INTERFACE I_StepCondition

PROPERTY getValue : BOOL
GET
END_GET
END_PROPERTY

PROPERTY isNegative : Bool
GET
END_GET
END_PROPERTY

PROPERTY isPositive : Bool
GET
END_GET
END_PROPERTY

METHOD NegCondition : BOOL
VAR_INPUT
END_VAR
END_METHOD

METHOD PosCondition : BOOL
VAR_INPUT
END_VAR
END_METHOD

PROPERTY setValue : Bool
SET
END_SET
END_PROPERTY

END_INTERFACE

(* stored: Version 1.1.0.1, ProductVersion 3.1.4024.2
   Itf I_StepCondition: Id {f45c417b-68ad-4c0b-a126-3513c0ea3d19}
   Property getValue: Id {7b981ae6-3b99-4c83-942d-56104da4fffc}
   Get Get: Id {8abdf485-509b-48f2-8800-a75dc7f05f5e}
   Property isNegative: Id {13870072-1c74-40a8-90bd-daee89c8b6bf}
   Get Get: Id {95b994b8-f6c6-442e-b7fb-18c2e592ac3c}
   Property isPositive: Id {b4cb559f-8319-4782-b92c-8fc776523afa}
   Get Get: Id {ac731e93-1ac9-4f40-bd2e-a6d303b4c552}
   Method NegCondition: Id {f84c5ef2-e96d-45c6-bc06-cdf8b894819a}
   Method PosCondition: Id {b9504ef5-21f3-436c-b0db-a7b273ebb7b4}
   Property setValue: Id {6923ac5c-b313-4703-97f2-d0ab16e525c6}
   Set Set: Id {97471d9e-d88e-451e-bd32-9c86b92b9898} *)
